PROGRAM MAIN
VAR
	fbCamera			:	FB_VN_SimpleCameraControl;
	eState				:	ETcVnCameraState;	

	fbAdaptiveThreshold: AdaptiveThreshold();
	fbBlobDecect: BlobDecect();
END_VAR

//fbAdaptiveThreshold(fbCamera:=fbCamera,eState:=eState);
fbBlobDecect(fbCamera:=fbCamera,eState:=eState);

END_PROGRAM

(* stored: Version 1.1.0.1, ProductVersion 3.1.4024.12
   POU MAIN: Id {21d0e6a1-4b68-4115-8f8e-5eae572fdde2}, SpecialFunc None *)
